Staubli VAL3: send2NextRob.pgx

program send2NextRob(num x_nConvNum (dimensions=1), num x_nID (dimensions=1), trsf x_trTrsf (dimensions=1), num x_nLatchedValue (dimensions=1))
begin
  // This program pushes an object into the transfer queue.
  // The production cycle pushes the objects to be transferred to
  //  the next robot into the transfer queue, and the tasks
  //  transferQueue will actually take care of sending the object
  //  to the next robot.
  //
  // Input parameters
  //  x_nConvNum      : Conveyor number
  //  x_nID           : ID of the object
  //  x_trTrsf        : Transformation of the object
  //  x_nLatchedValue : Latched encoder value of the object
  //
  // Output parameters
  //  None            :
  //
  //----------------------------------------------------------------
  //
  // If the ID of the next element of the queue is equals to -1, it
  //  means that the element is free and a new object can be stacked.
  //  Otherwise the queue is full.
  if _oTransferQueue[x_nConvNum,_nPushIndexTQ[x_nConvNum]].nID==-1
    _oTransferQueue[x_nConvNum,_nPushIndexTQ[x_nConvNum]].nLatchedValue=x_nLatchedValue
    _oTransferQueue[x_nConvNum,_nPushIndexTQ[x_nConvNum]].trTrsf=x_trTrsf
    // The last value updated is the ID. The task transferQueue is
    //  looking to this value in order to know if there is an object
    //  to be sent to the next robot.
    _oTransferQueue[x_nConvNum,_nPushIndexTQ[x_nConvNum]].nID=x_nID
    _nPushIndexTQ[x_nConvNum]=(_nPushIndexTQ[x_nConvNum]+1)%size(_oTransferQueue,2)
  else
    popUpMsg("Part not queued, transfer queue "+toString("",x_nConvNum+1)+" full")
  endIf
end
